// TwinCAT 3 PLC project MotorPLC
// ProgramVersion: 3.1.4024.0
// libraries:
//   Tc2_Standard, * (Beckhoff Automation GmbH)
//   Tc2_System, * (Beckhoff Automation GmbH)
//   Tc3_Module, * (Beckhoff Automation GmbH)
// project tree:
//   / PlcTask.TcTTO
//   POUs/ CoolingWaterValve.TcPOU, Encoder.TcPOU, Fan.TcPOU, HMI.TcPOU, MAIN.TcPOU, Motor.TcPOU, MotorProtection.TcPOU, Thermostat.TcPOU
// real-time tasks:
//   TASK PlcTask: cycle T#10ms, priority 20, ADS port 350

CONFIGURATION MotorPLC
    RESOURCE PLC ON TwinCAT3
        TASK PlcTask(INTERVAL := T#10ms, PRIORITY := 20);
        PROGRAM MAIN WITH PlcTask : MAIN;
    END_RESOURCE
END_CONFIGURATION

// ---- POUs/MAIN.TcPOU
PROGRAM MAIN
VAR
END_VAR

METHOD FB_init : BOOL
VAR_INPUT
	bInitRetains : BOOL; // if TRUE, the retain variables are initialized (warm start / cold start)
	bInCopyCode : BOOL;  // if TRUE, the instance afterwards gets moved into the copy code (online change)
END_VAR
END_METHOD

END_PROGRAM

// ---- POUs/CoolingWaterValve.TcPOU
FUNCTION_BLOCK CoolingWaterValve
VAR_INPUT
END_VAR
VAR_OUTPUT
END_VAR
VAR
	wOutputAddress AT %Q*: WORD;
	iPositionSetpoint : INT;
	rTemperatureSetpoint : REAL;
	rTemperatureActual : REAL := Thermostat.temperature;
END_VAR

METHOD FB_init : BOOL
VAR_INPUT
	bInitRetains : BOOL; // if TRUE, the retain variables are initialized (warm start / cold start)
	bInCopyCode : BOOL;  // if TRUE, the instance afterwards gets moved into the copy code (online change)
	
	
END_VAR
END_METHOD

METHOD setPosition : REAL
VAR_INPUT
END_VAR
END_METHOD

METHOD unscaleSetPosition : INT
VAR_INPUT
END_VAR
END_METHOD

END_FUNCTION_BLOCK

// ---- POUs/Thermostat.TcPOU
FUNCTION_BLOCK Thermostat
VAR_INPUT
END_VAR
VAR_OUTPUT
END_VAR
VAR
	wInputAddress AT %I* : WORD;
	rScaleMax : REAL;
	rScaleMin : REAL;
	iTemperatureAnalogValue : INT;
	rTemperatureScaledValue : REAL;
END_VAR

METHOD FB_init : BOOL
VAR_INPUT
	bInitRetains : BOOL; // if TRUE, the retain variables are initialized (warm start / cold start)
	bInCopyCode : BOOL;  // if TRUE, the instance afterwards gets moved into the copy code (online change)
END_VAR
END_METHOD

METHOD PRIVATE scaleTemperature : REAL
VAR_INPUT
END_VAR
END_METHOD

PROPERTY PUBLIC temperature : REAL
GET
temperature := rTemperatureScaledValue;
END_GET
END_PROPERTY

END_FUNCTION_BLOCK

// ---- POUs/Encoder.TcPOU
FUNCTION_BLOCK Encoder
VAR_INPUT
END_VAR
VAR_OUTPUT
END_VAR
VAR
	wDeviceAddress : WORD;
	iPositionActual : INT;
	iSpeedActual : INT;
END_VAR

METHOD FB_init : BOOL
VAR_INPUT
	bInitRetains : BOOL; // if TRUE, the retain variables are initialized (warm start / cold start)
	bInCopyCode : BOOL;  // if TRUE, the instance afterwards gets moved into the copy code (online change)
END_VAR
END_METHOD

PROPERTY PUBLIC positionActual : INT
GET
positionActual := iPositionActual;
END_GET
END_PROPERTY

PROPERTY PUBLIC speedActual : INT
GET
speedActual := iSpeedActual;
END_GET
END_PROPERTY

END_FUNCTION_BLOCK

// ---- POUs/Fan.TcPOU
FUNCTION_BLOCK Fan
VAR_INPUT
END_VAR
VAR_OUTPUT
END_VAR
VAR
	xOutputAddress AT %I* : BIT;
	bPowerStatus : BOOL;
END_VAR

METHOD FB_init : BOOL
VAR_INPUT
	bInitRetains : BOOL; // if TRUE, the retain variables are initialized (warm start / cold start)
	bInCopyCode : BOOL;  // if TRUE, the instance afterwards gets moved into the copy code (online change)
END_VAR
END_METHOD

METHOD powerOff : BOOL
VAR_INPUT
END_VAR
END_METHOD

METHOD powerOn : BOOL
VAR_INPUT
END_VAR
END_METHOD

PROPERTY PUBLIC powerStatus : BOOL
GET
powerStatus := bPowerStatus;
END_GET
END_PROPERTY

END_FUNCTION_BLOCK

// ---- POUs/HMI.TcPOU
FUNCTION_BLOCK HMI
VAR_INPUT
END_VAR
VAR_OUTPUT
END_VAR
VAR
	wDeviceAddress : WORD;
	wMotorAddress : WORD;
	bMotorPower : BOOL;
	bMotorOvercurrent : BOOL;
	rMotorTemperature : REAL;
	rMotorSpeed : REAL;
	rMotorPosition : REAL;
END_VAR

METHOD displayValues
VAR_INPUT
END_VAR
END_METHOD

METHOD FB_init : BOOL
VAR_INPUT
	bInitRetains : BOOL; // if TRUE, the retain variables are initialized (warm start / cold start)
	bInCopyCode : BOOL;  // if TRUE, the instance afterwards gets moved into the copy code (online change)
END_VAR
END_METHOD

METHOD writeValuesToDevice : BOOL
VAR_INPUT
END_VAR
END_METHOD

END_FUNCTION_BLOCK

// ---- POUs/Motor.TcPOU
FUNCTION_BLOCK Motor
VAR_INPUT
END_VAR
VAR_OUTPUT
END_VAR
VAR
	wDeviceAddress : WORD;
	rSpeedActual : REAL;
	rTorqueActual: REAL;
	rCurrentActual : REAL;
	rSpeedSetpoint : REAL;
	rTorqueSetpoint : REAL;
	bPowerStatus : BOOL;
	wErrorStatus : WORD;
END_VAR

PROPERTY PUBLIC currentActual : REAL
GET
currentActual := rCurrentActual;
END_GET
END_PROPERTY

PROPERTY PUBLIC errorStatus : WORD
GET
errorStatus := wErrorStatus;
END_GET
END_PROPERTY

METHOD FB_init : BOOL
VAR_INPUT
	bInitRetains : BOOL; // if TRUE, the retain variables are initialized (warm start / cold start)
	bInCopyCode : BOOL;  // if TRUE, the instance afterwards gets moved into the copy code (online change)
END_VAR
END_METHOD

PROPERTY PUBLIC powerStatus : BOOL
GET
powerStatus := bPowerStatus;
END_GET
END_PROPERTY

METHOD PUBLIC setSpeedSetpoint : BOOL
VAR_INPUT
END_VAR
END_METHOD

METHOD PUBLIC setTorqueSetpoint : BOOL
VAR_INPUT
END_VAR
END_METHOD

PROPERTY PUBLIC speedActual : REAL
GET
speedActual := rSpeedActual;
END_GET
END_PROPERTY

METHOD start : BOOL
VAR_INPUT
END_VAR
END_METHOD

METHOD stop : BOOL
VAR_INPUT
END_VAR
END_METHOD

PROPERTY PUBLIC torqueActual : REAL
GET
torqueActual := rTorqueActual;
END_GET
END_PROPERTY

END_FUNCTION_BLOCK

// ---- POUs/MotorProtection.TcPOU
FUNCTION_BLOCK MotorProtection
VAR_INPUT
END_VAR
VAR_OUTPUT
END_VAR
VAR
	xInputAddress AT %I* : BIT;
	bOvercurrentStatus : BOOL;
END_VAR

METHOD FB_init : BOOL
VAR_INPUT
	bInitRetains : BOOL; // if TRUE, the retain variables are initialized (warm start / cold start)
	bInCopyCode : BOOL;  // if TRUE, the instance afterwards gets moved into the copy code (online change)
END_VAR
END_METHOD

PROPERTY PUBLIC overcurrentStatus : BOOL
GET
overcurrentStatus := bOvercurrentStatus;
END_GET
END_PROPERTY

END_FUNCTION_BLOCK
